TYPE ST_AWEA_In :
STRUCT
	DoorOpened			:BIT;
	DoorClosed			:BIT;
	ProgReady			:BIT;
	ProgRun				:BIT;
	ProgEnd				:BIT;
	NotError			:BIT;
	Mode				:BIT;
	M401				:BIT;
	M402				:BIT;
	M403				:BIT;
END_STRUCT
END_TYPE

(* stored: Version 1.1.0.1, ProductVersion 3.1.4024.11
   DUT ST_AWEA_In: Id {6c1c00c0-8210-4461-b392-8b60cb936def} *)
